Omron Sysmac Studio project ExampleOpcUaRingBuffer (Sysmac Studio 1.63.0.7, StandardProject)

# Controller Example: NX102-9000 version 1.64
Task Services (priority 18, period or condition 4000): Models
Library RingBufferLib 0.0.2 (contents left out)
Library RingBufferOpcUaExtensionLib 0.0.2 (contents left out)

PROGRAM README
RETURN;
(*

# About this project
This project is an example project for `RingBufferOpcUaExtensionLib`.

## About the programs

* POU/Program/Models
This is a server-side program that exposes `RingBuffer` and performs remote operations.


# このプロジェクトについて
このプロジェクトは、`RingBufferOpcUaExtensionLib`の例示用プロジェクトです。

## プログラムについて

* POU/プログラム/Models
  `RingBuffer`を公開し、リモートからの操作を実行するサーバ側プログラムです。


For the parts to which I have rights, I follow POU/Program/LICENSE.
You are free to use and modify it, but we are not responsible for any damage or loss related to it.

(c) 2025 KITA Munemitsu

*)
END_PROGRAM

PROGRAM Models
VAR
    LoggerBuffer : stfreakjp\buf\extension\OpcUaRingBuffer;
    iBuffer : ARRAY[0..65534] OF BYTE;
    iBufferContext : stfreakjp\buf\RingBufferContext;
    iBinStr : ARRAY[0..255] OF BYTE;
    iBinStrSize : UINT;
    iInterval : UINT;
    iWaitTick : UINT;
END_VAR
IF P_First_Run THEN
	LoggerBuffer.Enable := TRUE;
	
	\\stfreakjp\buf\RingBuffer_init(
						Context:=iBufferContext,
						Buffer:=iBuffer);
	
	iWaitTick := 1;
	iInterval := iWaitTick;
END_IF;

Dec(iWaitTick);
IF iWaitTick < 1 THEN
	iBinStrSize
		:= StringToAry(In:=CONCAT('server=', DtToString(GetTime()), '$L'),
					   AryOut:=iBinStr[0]);
	\\stfreakjp\buf\RingBuffer_write(
						Context:=iBufferContext,
						Buffer:=iBuffer,
						In:=iBinStr,
						Head:=0,
						Size:=iBinStrSize,
						AllowOverWrite:=TRUE);
	iWaitTick := iInterval;
END_IF;

LoggerBuffer(BufferContext:=iBufferContext,
			 Buffer:=iBuffer);
END_PROGRAM

PROGRAM LICENSE
RETURN;
(*
The MIT License (MIT)

Copyright(c) 2025 KITA Munemitsu

Permission is hereby granted, free of charge, to any person obtaining a copy of this software and associated
documentation files (the “Software”), to deal in the Software without restriction, including without limitation
the rights to use, copy, modify, merge, publish, distribute, sublicense, and/or sell copies of the Software,
and to permit persons to whom the Software is furnished to do so, subject to the following conditions:

The above copyright notice and this permission notice shall be included in all copies or substantial portions of the Software.

THE SOFTWARE IS PROVIDED “AS IS”, WITHOUT WARRANTY OF ANY KIND, EXPRESS OR IMPLIED, INCLUDING BUT NOT
LIMITED TO THE WARRANTIES OF MERCHANTABILITY, FITNESS FOR A PARTICULAR PURPOSE AND NONINFRINGEMENT.
IN NO EVENT SHALL THE AUTHORS OR COPYRIGHT HOLDERS BE LIABLE FOR ANY CLAIM, DAMAGES OR OTHER LIABILITY,
WHETHER IN AN ACTION OF CONTRACT, TORT OR OTHERWISE, ARISING FROM, OUT OF OR IN CONNECTION WITH THE SOFTWARE
OR THE USE OR OTHER DEALINGS IN THE SOFTWARE.
*)
END_PROGRAM